{attribute 'GeneratedUsingTerminal: KL1002'}
{attribute addProperty BoxType "KL1002"}
{attribute addProperty Description ""}
{attribute addProperty Physics ""}
{attribute addProperty Id "Channel_1AT %I*Channel_87C95E760Channel_2AT %I*Channel_87C95E760"}
{attribute addProperty CRC "3141065359"}
{attribute addProperty Size "0"}
TYPE KL1002_BB38DA8F :
STRUCT
	{attribute addProperty Name "Channel_1"}
	Channel_1 : Channel_87C95E76;
	{attribute addProperty Name "Channel_2"}
	Channel_2 : Channel_87C95E76;
END_STRUCT
END_TYPE

(* stored: Version 1.2.0.0, ProductVersion 3.1.4024.9
   DUT KL1002_BB38DA8F: Id {d1d6314e-c6be-4eb1-8f15-e0c3b18d8fd7} *)
